FUNCTION_BLOCK FB_InstruNearDetect
VAR_INPUT
END_VAR
VAR_OUTPUT
END_VAR
VAR
	m_instruNearCounts :INT :=0;
	m_InstruNearCountThres :INT :=50;
END_VAR

// check if instrument is near
METHOD run : BOOL
VAR_INPUT
	IOValue :UDINT;
END_VAR
//Instrument single   At installation--2#0*0*   not installation --2#1*1*  And Hall single --2#100 0000
IF (IOValue AND 10#64) = 64  THEN
	m_instruNearCounts := MIN( m_instruNearCounts +1,m_InstruNearCountThres);
ELSE
	m_instruNearCounts := 0;
END_IF

run := m_instruNearCounts >= m_InstruNearCountThres;
END_METHOD

END_FUNCTION_BLOCK

(* stored: Version 1.1.0.1, ProductVersion 3.1.4024.11
   POU FB_InstruNearDetect: Id {e4e1dacc-521a-469b-84a8-012afab50104}, SpecialFunc None
   Method run: Id {1d951b0c-1d83-4922-a321-3e4bfb66656a} *)
